// Mitsubishi GX Works2 project: Compare   PLC: Q03UDV

PROGRAM MAIN
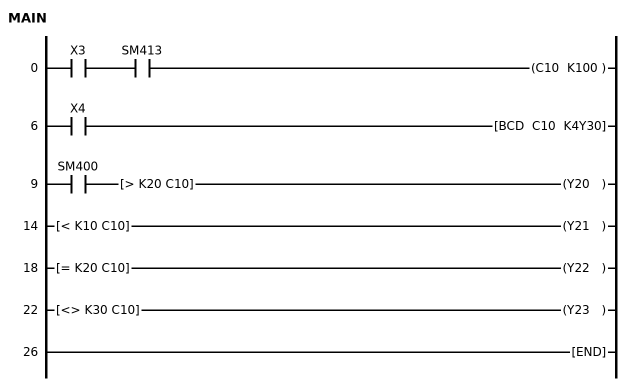
0     LD      X3
      AND     SM413
      OUT     C10 K100
6     LD      X4
      BCD     C10 K4Y30
9     LD      SM400
      AND>    K20 C10
      OUT     Y20
14    LD<     K10 C10
      OUT     Y21
18    LD=     K20 C10
      OUT     Y22
22    LD<>    K30 C10
      OUT     Y23
26    END
END_PROGRAM
